// TwinCAT 3 PLC project PLC
// Title: BaseClassExampleProgram
// Company: Red Rock Controls Limited
// Author: Roger Christopher
// ProjectVersion: 1.1.15.0
// Description: Updated to use tcl_BaseClasses V1.1.15.0
// ProgramVersion: 3.1.4023.0
// libraries:
//   Tc2_Standard, * (Beckhoff Automation GmbH)
//   Tc2_System, * (Beckhoff Automation GmbH)
//   Tc2_Utilities, * (Beckhoff Automation GmbH)
//   Tc3_Module, * (Beckhoff Automation GmbH)
//   tcl_BaseClasses, * (Red Rock Controls Limited)
//   VisuDialogs, * (System)
// project tree:
//   / GlobalTextList.TcGTLO, PlcTask.TcTTO, Visualization Manager.TcVMO (not stored)
//   GVLs/ DigitalInputs.TcGVL, DigitalOutputs.TcGVL, Globals.TcGVL, Notifications.TcGVL, Objects.TcGVL
//   POUs/Classes/Hmi Interface/ THmiInterface.TcPOU
//   POUs/Classes/Logger/ TLogger.TcPOU
//   POUs/Classes/Machine/ TMachine.TcPOU
//   POUs/Classes/Motor Starter/ TMotorStarter.TcPOU
//   POUs/Classes/Safety/ TSafety.TcPOU
//   POUs/ MAIN.TcPOU
//   POUs/Programs/ PB_Initialisation.TcPOU, PB_ObjectExecution.TcPOU
//   Version/ Global_Version.TcGVL
//   VISU/ Visualization.TcVIS
// real-time tasks:
//   TASK PlcTask: cycle T#10ms, priority 20, ADS port 350

CONFIGURATION PLC
    RESOURCE PLC ON TwinCAT3
        TASK PlcTask(INTERVAL := T#10ms, PRIORITY := 20);
        PROGRAM MAIN WITH PlcTask : MAIN;
    END_RESOURCE
END_CONFIGURATION

// ---- GVLs/DigitalInputs.TcGVL
{attribute 'qualified_only'}
VAR_GLOBAL
    EStopHealthy AT %I* : BOOL;
    StartPumpPb  AT %I* : BOOL;
END_VAR

// ---- GVLs/DigitalOutputs.TcGVL
{attribute 'qualified_only'}
VAR_GLOBAL
    HydraulicPumpRunningLamp  AT %Q* : BOOL;
END_VAR

// ---- GVLs/Globals.TcGVL
{attribute 'qualified_only'}
VAR_GLOBAL
    CurrentUserLoggedIn : BOOL;
    CurrentUserName     : STRING;
    CurrentUserAge      : INT;
    CurrentUserLevel    : UDINT;
    CurrentUserHeight   : LREAL;

END_VAR

// ---- GVLs/Notifications.TcGVL
{attribute 'qualified_only'}
VAR_GLOBAL
    
    // Global notification objects...
    Notification_OnUserLoggedIn  : T_Notification;
    Notification_OnUserLoggedOut : T_Notification;

END_VAR

// ---- GVLs/Objects.TcGVL
{attribute 'qualified_only'}
VAR_GLOBAL
    Machine            : TMachine;
    Safety             : TSafety;
    HmiInterface       : THmiInterface;
    Logging            : TLogger;
    HydraulicPumpMotor : TMotorStarter;
END_VAR

// ---- Version/Global_Version.TcGVL
{attribute 'TcGenerated'}
{attribute 'no-analysis'}
{attribute 'linkalways'}
// This function has been automatically generated from the project information.
VAR_GLOBAL CONSTANT
	{attribute 'const_non_replaced'}
	stLibVersion_BaseClassExampleProgram : ST_LibVersion := (iMajor := 1, iMinor := 1, iBuild := 15, iRevision := 0, nFlags := 0, sVersion := '1.1.15.0');
END_VAR

// ---- POUs/MAIN.TcPOU
PROGRAM MAIN
VAR
END_VAR

PB_Initialisation();
PB_ObjectExecution();

END_PROGRAM

// ---- POUs/Programs/PB_Initialisation.TcPOU
PROGRAM PB_Initialisation
VAR
    Initialised : BOOL;
    OnlineChangeCount : UDINT := 999;
END_VAR

IF NOT Initialised OR _AppInfo.OnlineChangeCnt <> OnlineChangeCount THEN
    // Re-link notification handlers...
    LinkNotificationHandlers();
    Initialised := TRUE;
    OnlineChangeCount := _AppInfo.OnlineChangeCnt;
END_IF

METHOD LinkNotificationHandlers
Objects.Safety.EStopTripped
    .ClearNotificationHandlers()
    .AddNotificationHandler(Objects.Machine.NotificationHandler_OnEstopTripped)
    .AddNotificationHandler(Objects.HydraulicPumpMotor.NotificationHandler_OnEstopTripped);

Objects.Safety.EStopReset
    .ClearNotificationHandlers()
    .AddNotificationHandler(Objects.Machine.NotificationHandler_OnEstopReset)
    .AddNotificationHandler(Objects.HydraulicPumpMotor.NotificationHandler_OnEstopReset);

// Notifications declared in the base class library, raised by all instances of T_Execution  
tcl_BaseClasses.GlobalNotifications.Notification_ExecutionAborted
    .ClearNotificationHandlers()
    .AddNotificationHandler(Objects.Logging.NotificationHandler_OnExecutionAborted);

tcl_BaseClasses.GlobalNotifications.Notification_ExecutionFailed
    .ClearNotificationHandlers()
    .AddNotificationHandler(Objects.Logging.NotificationHandler_OnExecutionFailed);

// Notification handlers accessed via properties...    
Notifications.Notification_OnUserLoggedIn
    .ClearNotificationHandlers()
    .AddNotificationHandler(Objects.Logging.NotificationHandler_OnUserLoggedIn);

Notifications.Notification_OnUserLoggedOut
    .ClearNotificationHandlers()
    .AddNotificationHandler(Objects.Logging.NotificationHandler_OnUserLoggedOut);
END_METHOD

END_PROGRAM

// ---- POUs/Programs/PB_ObjectExecution.TcPOU
PROGRAM PB_ObjectExecution
VAR
END_VAR

Objects.Machine(StartPb      := DigitalInputs.StartPumpPb,
                RunPumpMotor := Objects.HydraulicPumpMotor.RunMotor);

Objects.HydraulicPumpMotor(Running      => DigitalOutputs.HydraulicPumpRunningLamp);

Objects.Safety(EStopHealthy := DigitalInputs.EStopHealthy);

Objects.HmiInterface();

Objects.Logging();

END_PROGRAM

// ---- POUs/Classes/Machine/TMachine.TcPOU
FUNCTION_BLOCK TMachine
VAR_INPUT
    StartPb          : BOOL;
    RunPumpMotor : I_Execution; // Machine controls the pump motor, but does not own it
END_VAR
VAR
    EnablePower : BOOL;

    Starting       : BOOL;
    Running        : BOOL;
    
    RisingEdge_StartPbPressed : T_RisingEdge;

    NotificationHandler_OnEstopReset   : T_NotificationHandler;
    NotificationHandler_OnEstopTripped : T_NotificationHandler;
END_VAR

HandleNotifications();

IF RisingEdge_StartPbPressed.Test(StartPb) THEN
    F_LogMessage('Machine', 'Start PB pressed');
    IF EnablePower THEN
        RunPumpMotor.Start();
        Starting := TRUE;
    ELSE
        F_LogWarning('Machine','Cannot start pump - power not enabled');
    END_IF
END_IF

IF Starting THEN
    IF RunPumpMotor.Done THEN
        Starting := FALSE;
        Running  := TRUE;
    END_IF
    IF RunPumpMotor.Error THEN
        Starting := FALSE;
        Running  := FALSE;
    END_IF

END_IF

METHOD HandleNotifications
VAR_INPUT
END_VAR
IF NotificationHandler_OnEstopReset.IsRaised() THEN
    OnEStopReset();
END_IF

IF NotificationHandler_OnEstopTripped.IsRaised() THEN
    OnEStopTripped();
END_IF
END_METHOD

METHOD OnEStopReset
EnablePower := TRUE;
F_LogError(Source  := 'Machine',
           Message := 'EStop was reset');
END_METHOD

METHOD OnEStopTripped
EnablePower := FALSE;
Running     := FALSE;

F_LogError(Source  := 'Machine',
           Message := 'EStop was tripped');
END_METHOD

END_FUNCTION_BLOCK

// ---- POUs/Classes/Safety/TSafety.TcPOU
FUNCTION_BLOCK TSafety
VAR_INPUT
    EStopHealthy : BOOL;
END_VAR
VAR
    RisingEdge_EStopHealthy : T_RisingEdge;
    FallingEdge_EStopHealthy    : T_FallingEdge;

    // Local notification objects...
    EStopTripped : T_Notification;
    EStopReset   : T_Notification;
END_VAR

IF RisingEdge_EStopHealthy.Test(EStopHealthy) THEN
    EStopReset.Raise();
END_IF

IF FallingEdge_EStopHealthy.Test(EStopHealthy) THEN
    EStopTripped.Raise();
END_IF

END_FUNCTION_BLOCK

// ---- POUs/Classes/Hmi Interface/THmiInterface.TcPOU
FUNCTION_BLOCK THmiInterface
VAR
    // Data set via the Hmi...
    LogIn      : BOOL;
    LogOut     : BOOL;
    
    UserName   : STRING := 'Horatio';
    UserAge    : INT    := 23;
    UserLevel  : UDINT  := 999;
    UserHeight : LREAL  := 1.80;

    RisingEdge_LogIn  : T_RisingEdge;
    RisingEdge_LogOut  : T_RisingEdge;

END_VAR

IF RisingEdge_LogIn.Test(LogIn) THEN
    // set the event args...
    Notifications.Notification_OnUserLoggedIn.Args
        .Add_STRING(UserName)
        .Add_INT(UserAge)
        .Add_UDINT(UserLevel)
        .Add_LREAL(UserHeight);

    // ...then raise the event
    Notifications.Notification_OnUserLoggedIn.Raise();

END_IF

IF RisingEdge_LogOut.Test(LogOut) THEN
    Notifications.Notification_OnUserLoggedOut.Raise();
END_IF

END_FUNCTION_BLOCK

// ---- POUs/Classes/Logger/TLogger.TcPOU
FUNCTION_BLOCK TLogger
VAR
    _NotificationHandler_OnUserLoggedIn     : T_NotificationHandler;
    _NotificationHandler_OnUserLoggedOut    : T_NotificationHandler;
    _NotificationHandler_OnExecutionAborted : T_NotificationHandler;
    _NotificationHandler_OnExecutionFailed  : T_NotificationHandler;

END_VAR

HandleNotifications();

METHOD HandleNotifications
VAR_INPUT
END_VAR
IF _NotificationHandler_OnExecutionFailed.IsRaised() THEN
    F_LogError(Source  := 'T_Execution',
               Message := _NotificationHandler_OnExecutionFailed.Args.Read_STRING());
END_IF

IF _NotificationHandler_OnExecutionAborted.IsRaised() THEN
    F_LogError(Source  := 'T_Execution',
               Message := _NotificationHandler_OnExecutionAborted.Args.Read_STRING());
END_IF

IF _NotificationHandler_OnUserLoggedIn.IsRaised() THEN
    IF NOT Globals.CurrentUserLoggedIn THEN
        Globals.CurrentUserLoggedIn := TRUE;

        Globals.CurrentUserName   := _NotificationHandler_OnUserLoggedIn.Args.Read_STRING();
        Globals.CurrentUserAge    := _NotificationHandler_OnUserLoggedIn.Args.Read_INT();
        Globals.CurrentUserLevel  := _NotificationHandler_OnUserLoggedIn.Args.Read_UDINT();
        Globals.CurrentUserHeight := _NotificationHandler_OnUserLoggedIn.Args.Read_LREAL();

        F_LogError(Source  := 'Logging',
                   Message := 'User logged in');
    END_IF
END_IF

IF _NotificationHandler_OnUserLoggedOut.IsRaised() THEN
    IF Globals.CurrentUserLoggedIn THEN
        Globals.CurrentUserLoggedIn := FALSE;

        Globals.CurrentUserName   := '';
        Globals.CurrentUserAge    := 0;
        Globals.CurrentUserLevel  := 999;
        Globals.CurrentUserHeight := 0.0;

        F_LogError(Source  := 'Logging',
                   Message := 'User logged out');
    END_IF
END_IF
END_METHOD

PROPERTY NotificationHandler_OnExecutionAborted : I_NotificationHandler
GET
NotificationHandler_OnExecutionAborted := _NotificationHandler_OnExecutionAborted;
END_GET
END_PROPERTY

PROPERTY NotificationHandler_OnExecutionFailed : I_NotificationHandler
GET
NotificationHandler_OnExecutionFailed := _NotificationHandler_OnExecutionFailed;
END_GET
END_PROPERTY

PROPERTY NotificationHandler_OnUserLoggedIn : I_NotificationHandler
GET
NotificationHandler_OnUserLoggedIn := _NotificationHandler_OnUserLoggedIn;
END_GET
END_PROPERTY

PROPERTY NotificationHandler_OnUserLoggedOut : I_NotificationHandler
GET
NotificationHandler_OnUserLoggedOut := _NotificationHandler_OnUserLoggedOut;
END_GET
END_PROPERTY

END_FUNCTION_BLOCK

// ---- POUs/Classes/Motor Starter/TMotorStarter.TcPOU
FUNCTION_BLOCK TMotorStarter
VAR_INPUT
END_VAR
VAR_OUTPUT
    Running : BOOL;
END_VAR
VAR
    _RunMotor  : T_Execution;
    EStopHealthy : BOOL;
    Run        : BOOL;
    ErrorMsg   : STRING;
    OnTimer_RunMotor       : T_OnTimer(2.0);
    
    NotificationHandler_OnEstopReset   : T_NotificationHandler;
    NotificationHandler_OnEstopTripped : T_NotificationHandler;
END_VAR

HandleNotifications();

IF _RunMotor.Starting THEN
    _RunMotor.SetBusy();
    Run   := TRUE;
END_IF
IF RunMotor.Busy AND Running THEN
    F_LogMessage('Motor Starter', 'Motor has started');
    _RunMotor.SetDone();
END_IF
IF RunMotor.Busy AND NOT EStopHealthy THEN
     ErrorMsg := 'Cannot start motor - EStop tripped';
    _RunMotor.SetError(ErrorMsg);
END_IF
IF _RunMotor.Aborting THEN
    Run   := FALSE;
    _RunMotor.SetAborted();
END_IF

// Simulate motor starting...
Running := OnTimer_RunMotor.Delay(Run);

METHOD HandleNotifications
VAR_INPUT
END_VAR
IF NotificationHandler_OnEstopReset.IsRaised() THEN
    EStopHealthy := TRUE;
END_IF

IF NotificationHandler_OnEstopTripped.IsRaised() THEN
    EStopHealthy := FALSE;
    Run := FALSE;
END_IF
END_METHOD

PROPERTY RunMotor : I_Execution
GET
RunMotor := _RunMotor;
END_GET
END_PROPERTY

END_FUNCTION_BLOCK

// ---- GlobalTextList.TcGTLO
TEXTLIST GlobalTextList
  545 = '  %.2 m'
  613 = '  %.2f m'
  367 = '  %d'
  771 = '  %s'
  759 = 'Age'
  136 = 'Current User'
  561 = 'EStop Healthy'
  639 = 'Height'
  33 = 'Hydraulic Pump Running'
  902 = 'Log In'
  204 = 'Log In Dialog'
  966 = 'Log Out'
  939 = 'Name'
  953 = 'Pump Running'
  418 = 'Running'
  171 = 'Start PB'
  709 = 'Start Pump'
  691 = 'User Level'
  742 = 'User Name'
  542 = 'Username'
END_TEXTLIST

// ---- VISU/Visualization.TcVIS
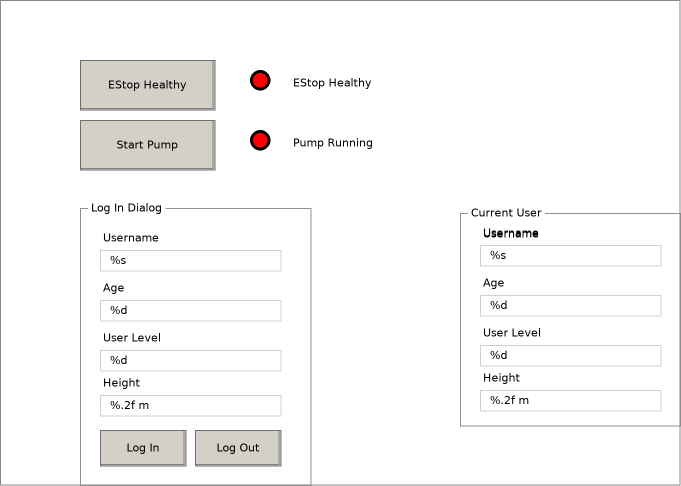
VISUALIZATION Visualization  // 681x486
    Button (80,60 135x50), "EStop Healthy"
        toggle DigitalInputs.EStopHealthy
    Button (80,120 135x50), "Start Pump"
        tap DigitalInputs.StartPumpPb
    Ellipse (250,130 20x20), colour toggle: DigitalOutputs.HydraulicPumpRunningLamp
    Label (290,135 151x16), "Pump Running"
    Ellipse (250,70 20x20), colour toggle: DigitalInputs.EStopHealthy
    Label (290,75 151x16), "EStop Healthy"
    GroupBox (80,200 231x286), "Log In Dialog"
        Textfield (20,50 181x21), "%s", text variable: Objects.HmiInterface.UserName
            OnMouseClick: write the text variable via Default
        Label (20,80 151x16), "Age"
        Textfield (20,100 181x21), "%d", text variable: Objects.HmiInterface.UserAge
            OnMouseClick: write the text variable via Default
        Label (20,130 151x16), "User Level"
        Textfield (20,150 181x21), "%d", text variable: Objects.HmiInterface.UserLevel
            OnMouseClick: write the text variable via Default
        Label (20,175 151x16), "Height"
        Textfield (20,195 181x21), "%.2f m", text variable: Objects.HmiInterface.UserHeight
            OnMouseClick: write the text variable via Default
        Button (20,230 86x36), "Log In"
            tap Objects.HmiInterface.LogIn
        Button (115,230 86x36), "Log Out"
            tap Objects.HmiInterface.LogOut
        Label (400,25 151x16), "Username"
        Label (20,30 151x16), "Username"
    GroupBox (460,205 221x221), "Current User"
        Label (20,21 151x16), "Username"
    Textfield (480,245 181x21), "%s", text variable: Globals.CurrentUserName
    Label (480,275 151x16), "Age"
    Textfield (480,295 181x21), "%d", text variable: Globals.CurrentUserAge
    Label (480,325 151x16), "User Level"
    Textfield (480,345 181x21), "%d", text variable: Globals.CurrentUserLevel
    Label (480,370 151x16), "Height"
    Textfield (480,390 181x21), "%.2f m", text variable: Globals.CurrentUserHeight
END_VISUALIZATION
